// TIA Portal project "scl_asenkron_motor" (V18)

(* hardware
DEVICE "S7-1200 station_1"  S7-1200 Station
   slot 0: "Rack_0"  S7-1200 Rack  Rack  V1.0
   slot 1: "PLC_1"  CPU 1214C DC/DC/DC  6ES7 214-1AG40-0XB0  V4.6
*)

// ===== PLC "PLC_1"  CPU 1214C DC/DC/DC =====

VAR_GLOBAL   // PLC tag table "Default tag table"
   "STOP" AT %I0.0 : Bool;
   "AŞIRI AKIM" AT %I0.1 : Bool;
   "İLERİ START" AT %I0.2 : Bool;
   "GERİ START" AT %I0.3 : Bool;
   "İLERİ RÖLE" AT %Q0.0 : Bool;
   "GERİ RÖLE" AT %Q0.1 : Bool;
END_VAR

FUNCTION "Block_1" : Void   // FC1, SCL
{ S7_Optimized_Access := 'TRUE' }
VERSION : 0.1
BEGIN
   "İLERİ RÖLE" := ("İLERİ START" OR "İLERİ RÖLE") AND NOT "GERİ RÖLE";

   "GERİ RÖLE" := ("GERİ START" OR "GERİ RÖLE") AND NOT "İLERİ RÖLE";

   IF "STOP"=1 OR "AŞIRI AKIM"=1 THEN

       "İLERİ RÖLE" := 0;
       "GERİ RÖLE" := 0;
   END_IF;
END_FUNCTION

ORGANIZATION_BLOCK "Main"   // OB1, LAD, ProgramCycle
TITLE = "Main Program Sweep (Cycle)"
{ S7_Optimized_Access := 'TRUE' }
VERSION : 0.1
// UYGULAMA-1: 3 fazli asenkron motor ileri_buton ile ileri yönde, geri_buton" ile geri yönde
// çalistirlacaktir. "stop" butonu basilinca da duracaktir. Bir yönde çalisirken durdurulmadan diger
// yönde çalismayacaktir. Ayrica motor 'asir akim" rölesi (F2) ile korunacaktir.
   VAR_INPUT
      Initial_Call : Bool;   // Initial call of this OB
      Remanence : Bool;   // =True, if remanent data are available
   END_VAR
BEGIN
END_ORGANIZATION_BLOCK